PROGRAM Lamp
VAR
	countercounter : int;
END_VAR

countercounter := countercounter +1;

END_PROGRAM

(* stored: Version 1.1.0.1, ProductVersion 3.1.4024.12
   POU Lamp: Id {469f8485-acfa-458d-ac11-64caf7a17e5c}, SpecialFunc None *)
